SMOVL C00364 BC00364 V=166.7  +MOVJ EC00364
SREFP 3 C00365 BC00365  +REFP EC00365
CALL JOB:SEARCH-R1-S13D
SET P028 P006
SFTON3D P028
SMOVL C00366 BC00366 V=166.7  +MOVJ EC00366
SREFP 3 C00367 BC00367  +REFP EC00367
CALL JOB:SEARCH-R1-S13D
SET P028 P006
SFTON3D P028
SMOVL C00368 BC00368 V=250.0  +MOVJ EC00368
MOVL C00369 BC00369 V=1000.0  +MOVJ EC00369 VJ=100.00
'EndPath S4609
MOVJ C00370 BC00370 VJ=100.00  +MOVJ EC00370 VJ=100.00
'Path S4882
SFTOF3D
MOVJ C00371 BC00371 VJ=100.00  +MOVJ EC00371 VJ=100.00
MOVL C00372 BC00372 V=800.0  +MOVJ EC00372 VJ=100.00
SMOVL C00373 BC00373 V=166.7  +MOVJ EC00373
SREFP 3 C00374 BC00374  +REFP EC00374
CALL JOB:SEARCH-R1-S13D
SET P060 P006
SFTON3D P060
SMOVL C00375 BC00375 V=166.7  +MOVJ EC00375
SMOVL C00376 BC00376 V=166.7  +MOVJ EC00376
SREFP 3 C00377 BC00377  +REFP EC00377
CALL JOB:SEARCH-R1-S13D
SET P060 P006
SFTON3D P060
SMOVL C00378 BC00378 V=166.7  +MOVJ EC00378
SMOVL C00379 BC00379 V=333.3  +MOVJ EC00379
SMOVL C00380 BC00380 V=166.7  +MOVJ EC00380
SREFP 3 C00381 BC00381  +REFP EC00381
CALL JOB:SEARCH-R1-S13D
SET P060 P006
SFTON3D P060
SMOVL C00382 BC00382 V=166.7  +MOVJ EC00382
MOVL C00383 BC00383 V=1000.0  +MOVJ EC00383 VJ=100.00
'EndPath S4882
MOVJ C00384 BC00384 VJ=100.00  +MOVJ EC00384 VJ=100.00
COMM 'Path S4610
COMM PAUSE
COMM SFTOF3D
COMM MOVJ C00385 BC00385 VJ=100.00  +MOVJ EC00385 VJ=100.00
COMM MOVL C00386 BC00386 V=800.0  +MOVJ EC00386 VJ=100.00
COMM SMOVL C00387 BC00387 V=166.7  +MOVJ EC00387
COMM SREFP 3 C00388 BC00388  +REFP EC00388
COMM CALL JOB:SEARCH-R1-S13D
COMM SET P029 P006
COMM SFTON3D P029
COMM SMOVL C00389 BC00389 V=166.7  +MOVJ EC00389
COMM SREFP 3 C00390 BC00390  +REFP EC00390
COMM CALL JOB:SEARCH-R1-S13D
COMM SET P029 P006
COMM SFTON3D P029
COMM SMOVL C00391 BC00391 V=166.7  +MOVJ EC00391
COMM MOVL C00392 BC00392 V=1000.0  +MOVJ EC00392 VJ=100.00
COMM 'EndPath S4610
COMM 'Path S4611
COMM SFTOF3D
COMM MOVJ C00393 BC00393 VJ=100.00  +MOVJ EC00393 VJ=100.00
COMM MOVL C00394 BC00394 V=800.0  +MOVJ EC00394 VJ=100.00
COMM SMOVL C00395 BC00395 V=166.7  +MOVJ EC00395
COMM SREFP 3 C00396 BC00396  +REFP EC00396
COMM CALL JOB:SEARCH-R1-S13D
COMM SET P030 P006
COMM SFTON3D P030
COMM SMOVL C00397 BC00397 V=166.7  +MOVJ EC00397
COMM SREFP 3 C00398 BC00398  +REFP EC00398
COMM CALL JOB:SEARCH-R1-S13D
COMM SET P030 P006
COMM SFTON3D P030
COMM SMOVL C00399 BC00399 V=166.7  +MOVJ EC00399
COMM MOVL C00400 BC00400 V=800.0  +MOVJ EC00400 VJ=100.00
COMM MOVL C00401 BC00401 V=1000.0  +MOVJ EC00401 VJ=100.00
COMM 'EndPath S4611
MOVJ C00402 BC00402 VJ=100.00  +MOVJ EC00402 VJ=100.00
'Path S4612
SFTOF3D
MOVJ C00403 BC00403 VJ=100.00  +MOVJ EC00403 VJ=100.00
MOVL C00404 BC00404 V=800.0  +MOVJ EC00404 VJ=100.00
SMOVL C00405 BC00405 V=166.7  +MOVJ EC00405
SREFP 3 C00406 BC00406  +REFP EC00406
CALL JOB:SEARCH-R1-S13D
SET P031 P006
SFTON3D P031
SMOVL C00407 BC00407 V=166.7  +MOVJ EC00407
SMOVL C00408 BC00408 V=166.7  +MOVJ EC00408
SREFP 3 C00409 BC00409  +REFP EC00409
CALL JOB:SEARCH-R1-S13D
SET P031 P006
SFTON3D P031
SMOVL C00410 BC00410 V=166.7  +MOVJ EC00410
SMOVL C00411 BC00411 V=166.7  +MOVJ EC00411
SREFP 3 C00412 BC00412  +REFP EC00412
CALL JOB:SEARCH-R1-S13D
SET P031 P006
SFTON3D P031
SMOVL C00413 BC00413 V=166.7  +MOVJ EC00413
MOVL C00414 BC00414 V=1000.0  +MOVJ EC00414 VJ=100.00
'EndPath S4612
MOVJ C00415 BC00415 VJ=100.00  +MOVJ EC00415 VJ=100.00
'Path S4613
SFTOF3D
MOVJ C00416 BC00416 VJ=100.00  +MOVJ EC00416 VJ=100.00
MOVL C00417 BC00417 V=800.0  +MOVJ EC00417 VJ=100.00
SMOVL C00418 BC00418 V=166.7  +MOVJ EC00418
SREFP 3 C00419 BC00419  +REFP EC00419
CALL JOB:SEARCH-R1-S13D
SET P032 P006
SFTON3D P032
SMOVL C00420 BC00420 V=166.7  +MOVJ EC00420
SREFP 3 C00421 BC00421  +REFP EC00421
CALL JOB:SEARCH-R1-S13D
SET P032 P006
SFTON3D P032
SMOVL C00422 BC00422 V=166.7  +MOVJ EC00422
SMOVL C00423 BC00423 V=166.7  +MOVJ EC00423
SREFP 3 C00424 BC00424  +REFP EC00424
CALL JOB:SEARCH-R1-S13D
SET P032 P006
SFTON3D P032
SMOVL C00425 BC00425 V=166.7  +MOVJ EC00425
MOVL C00426 BC00426 V=1000.0  +MOVJ EC00426 VJ=100.00
'EndPath S4613
MOVJ C00427 BC00427 VJ=100.00  +MOVJ EC00427 VJ=100.00
'Path S4614
SFTOF3D
MOVJ C00428 BC00428 VJ=100.00  +MOVJ EC00428 VJ=100.00
MOVL C00429 BC00429 V=800.0  +MOVJ EC00429 VJ=100.00
SMOVL C00430 BC00430 V=166.7  +MOVJ EC00430
SREFP 3 C00431 BC00431  +REFP EC00431
CALL JOB:SEARCH-R1-S13D
SET P033 P006
SFTON3D P033
SMOVL C00432 BC00432 V=166.7  +MOVJ EC00432
SREFP 3 C00433 BC00433  +REFP EC00433
CALL JOB:SEARCH-R1-S13D
SET P033 P006
SFTON3D P033
SMOVL C00434 BC00434 V=166.7  +MOVJ EC00434
MOVL C00435 BC00435 V=1000.0  +MOVJ EC00435 VJ=100.00
'EndPath S4614
'Path S4615
SFTOF3D
MOVJ C00436 BC00436 VJ=100.00  +MOVJ EC00436 VJ=100.00
MOVL C00437 BC00437 V=800.0  +MOVJ EC00437 VJ=100.00
SMOVL C00438 BC00438 V=166.7  +MOVJ EC00438
SREFP 3 C00439 BC00439  +REFP EC00439
CALL JOB:SEARCH-R1-S13D
SET P034 P006
SFTON3D P034
SMOVL C00440 BC00440 V=166.7  +MOVJ EC00440
SREFP 3 C00441 BC00441  +REFP EC00441
CALL JOB:SEARCH-R1-S13D
SET P034 P006
SFTON3D P034
SMOVL C00442 BC00442 V=166.7  +MOVJ EC00442
SMOVL C00443 BC00443 V=166.7  +MOVJ EC00443
SREFP 3 C00444 BC00444  +REFP EC00444
CALL JOB:SEARCH-R1-S13D
SET P034 P006
SFTON3D P034
SMOVL C00445 BC00445 V=166.7  +MOVJ EC00445
MOVL C00446 BC00446 V=1000.0  +MOVJ EC00446 VJ=100.00
'EndPath S4615
MOVJ C00447 BC00447 VJ=100.00  +MOVJ EC00447 VJ=100.00
MOVJ C00448 BC00448 VJ=100.00  +MOVJ EC00448 VJ=100.00
'Path W4616
SFTOF3D
SFTON3D P026
MOVJ C00449 BC00449 VJ=100.00  +MOVJ EC00449 VJ=100.00
SMOVL C00450 BC00450 V=800.0  +MOVJ EC00450
'POPRAWIC!!!!
SMOVL C00451 BC00451 V=166.7 PL=0  +MOVJ EC00451
MACRO1 MJ#(0) ARGF21
ARCON
SWVON WEV#(100)
SMOVL C00452 BC00452 V=9.2  +MOVJ EC00452
SFTON3D P091
SMOVL C00453 BC00453 V=9.2  +MOVJ EC00453
SMOVL C00454 BC00454 V=9.2  +MOVJ EC00454
SWVOF
ARCOF
SMOVL C00455 BC00455 V=800.0  +MOVJ EC00455
SMOVL C00456 BC00456 V=1000.0  +MOVJ EC00456
SFTOF3D
'EndPath W4616
MOVJ C00457 BC00457 VJ=100.00  +MOVJ EC00457 VJ=100.00
'Path W4617
SFTOF3D
SFTON3D P028
MOVJ C00458 BC00458 VJ=100.00  +MOVJ EC00458 VJ=100.00
MOVJ C00459 BC00459 VJ=100.00  +MOVJ EC00459 VJ=100.00
SMOVL C00460 BC00460 V=800.0  +MOVJ EC00460
SMOVL C00461 BC00461 V=150.0 PL=0  +MOVJ EC00461
ARCON
SWVON WEV#(100)
MOVL C00462 BC00462 V=9.2  +MOVJ EC00462 VJ=100.00
SFTON3D P027
SMOVL C00463 BC00463 V=9.2  +MOVJ EC00463
SMOVL C00464 BC00464 V=9.2  +MOVJ EC00464
ARCOF
SWVOF
SMOVL C00465 BC00465 V=800.0  +MOVJ EC00465
SMOVL C00466 BC00466 V=1000.0  +MOVJ EC00466
SFTOF3D
'EndPath W4617
MOVJ C00467 BC00467 VJ=100.00  +MOVJ EC00467 VJ=100.00
'Path W4618
COMM PAUSE
COMM SFTOF3D
COMM SFTON3D P022
COMM MOVJ C00468 BC00468 VJ=100.00  +MOVJ EC00468 VJ=100.00
COMM SMOVL C00469 BC00469 V=800.0  +MOVJ EC00469
COMM SMOVL C00470 BC00470 V=150.0 PL=0  +MOVJ EC00470
COMM MACRO1 MJ#(0) ARGF9
COMM ARCON
COMM SWVON WEV#(60)
COMM SFTON3D P021
COMM SMOVL C00471 BC00471 V=10.0  +MOVJ EC00471
COMM ARCOF
COMM SWVOF
COMM SMOVL C00472 BC00472 V=800.0  +MOVJ EC00472
COMM SMOVL C00473 BC00473 V=1000.0  +MOVJ EC00473
COMM SFTOF3D
COMM 'EndPath W4618
COMM 'Path W4883
SFTOF3D
SFTON3D P060
MOVJ C00474 BC00474 VJ=100.00  +MOVJ EC00474 VJ=100.00
MACRO1 MJ#(0) ARGF9
SMOVL C00475 BC00475 V=800.0  +MOVJ EC00475
SMOVL C00476 BC00476 V=150.0 PL=0  +MOVJ EC00476
ARCON
SMOVL C00477 BC00477 V=10.0  +MOVJ EC00477
SMOVL C00478 BC00478 V=10.0  +MOVJ EC00478
SMOVL C00479 BC00479 V=10.0  +MOVJ EC00479
ARCOF
SMOVL C00480 BC00480 V=800.0  +MOVJ EC00480
SFTOF3D
'EndPath W4883
'Path W4884
SFTOF3D
SFTON3D P060
SMOVL C00481 BC00481 V=800.0  +MOVJ EC00481
SMOVL C00482 BC00482 V=150.0 PL=0  +MOVJ EC00482
ARCON
SMOVL C00483 BC00483 V=10.0  +MOVJ EC00483
SMOVL C00484 BC00484 V=10.0  +MOVJ EC00484
SMOVL C00485 BC00485 V=10.0  +MOVJ EC00485
ARCOF
SMOVL C00486 BC00486 V=800.0  +MOVJ EC00486
SMOVL C00487 BC00487 V=1000.0  +MOVJ EC00487
SFTOF3D
'EndPath W4884
MOVJ C00488 BC00488 VJ=100.00  +MOVJ EC00488 VJ=100.00
COMM 'Path W4619
COMM PAUSE
COMM SFTOF3D
COMM SFTON3D P030
COMM MOVJ C00489 BC00489 VJ=100.00  +MOVJ EC00489 VJ=100.00
COMM MOVJ C00490 BC00490 VJ=100.00  +MOVJ EC00490 VJ=100.00
COMM SMOVL C00491 BC00491 V=800.0  +MOVJ EC00491
COMM SMOVL C00492 BC00492 V=150.0 PL=0  +MOVJ EC00492
COMM ARCON
COMM MOVL C00493 BC00493 V=10.0  +MOVJ EC00493 VJ=100.00
COMM SFTON3D P029
COMM SMOVL C00494 BC00494 V=10.0  +MOVJ EC00494
COMM SMOVL C00495 BC00495 V=10.0  +MOVJ EC00495
COMM ARCOF
COMM SMOVL C00496 BC00496 V=800.0  +MOVJ EC00496
COMM SMOVL C00497 BC00497 V=1000.0  +MOVJ EC00497
COMM SFTOF3D
COMM 'EndPath W4619
MOVJ C00498 BC00498 VJ=100.00  +MOVJ EC00498 VJ=100.00
MOVJ C00499 BC00499 VJ=100.00  +MOVJ EC00499 VJ=100.00
'Path W4620
SFTOF3D
SFTON3D P033
MOVJ C00500 BC00500 VJ=100.00  +MOVJ EC00500 VJ=100.00
SMOVL C00501 BC00501 V=800.0  +MOVJ EC00501
SMOVL C00502 BC00502 V=166.7 PL=0  +MOVJ EC00502
ARCON
SMOVL C00503 BC00503 V=9.2  +MOVJ EC00503
SFTON3D P034
SMOVL C00504 BC00504 V=9.2  +MOVJ EC00504
SMOVL C00505 BC00505 V=9.2  +MOVJ EC00505
ARCOF
SMOVL C00506 BC00506 V=800.0  +MOVJ EC00506
SMOVL C00507 BC00507 V=1000.0  +MOVJ EC00507
SFTOF3D
'EndPath W4620
MOVJ C00508 BC00508 VJ=100.00  +MOVJ EC00508 VJ=100.00
'Path W4621
SFTOF3D
SFTON3D P024
MOVJ C00509 BC00509 VJ=100.00  +MOVJ EC00509 VJ=100.00
SMOVL C00510 BC00510 V=800.0  +MOVJ EC00510
SMOVL C00511 BC00511 V=166.7 PL=0  +MOVJ EC00511
ARCON
SMOVL C00512 BC00512 V=10.0  +MOVJ EC00512
SFTON3D P025
SMOVL C00513 BC00513 V=10.0  +MOVJ EC00513
SMOVL C00514 BC00514 V=10.0  +MOVJ EC00514
ARCOF
SMOVL C00515 BC00515 V=800.0  +MOVJ EC00515
SMOVL C00516 BC00516 V=1000.0  +MOVJ EC00516
SFTOF3D
'EndPath W4621
MOVJ C00517 BC00517 VJ=100.00  +MOVJ EC00517 VJ=100.00
MOVJ C00518 BC00518 VJ=100.00  +MOVJ EC00518 VJ=100.00
'Path W4622
SFTOF3D
SFTON3D P032
MOVJ C00519 BC00519 VJ=100.00  +MOVJ EC00519 VJ=100.00
SMOVL C00520 BC00520 V=800.0  +MOVJ EC00520
SMOVL C00521 BC00521 V=166.7 PL=0  +MOVJ EC00521
ARCON
SMOVL C00522 BC00522 V=9.2  +MOVJ EC00522
SFTON3D P031
SMOVL C00523 BC00523 V=9.2  +MOVJ EC00523
SMOVL C00524 BC00524 V=9.2  +MOVJ EC00524
ARCOF
SMOVL C00525 BC00525 V=800.0  +MOVJ EC00525
SMOVL C00526 BC00526 V=1000.0  +MOVJ EC00526
SFTOF3D
'EndPath W4622
'Path W4623
SFTOF3D
SFTON3D P023
MOVJ C00527 BC00527 VJ=100.00  +MOVJ EC00527 VJ=100.00
JUMP *VVP
MOVJ C00528 BC00528 VJ=100.00  +MOVJ EC00528 VJ=100.00
SMOVL C00529 BC00529 V=800.0  +MOVJ EC00529
SMOVL C00530 BC00530 V=166.7 PL=0  +MOVJ EC00530
'ARCON DO SPRAWDZENIA
PAUSE
SMOVL C00531 BC00531 V=10.0  +MOVJ EC00531
SMOVL C00532 BC00532 V=10.0  +MOVJ EC00532
SMOVL C00533 BC00533 V=10.0  +MOVJ EC00533
SMOVL C00534 BC00534 V=10.0  +MOVJ EC00534
SMOVL C00535 BC00535 V=10.0  +MOVJ EC00535
SMOVL C00536 BC00536 V=10.0  +MOVJ EC00536
SMOVL C00537 BC00537 V=10.0  +MOVJ EC00537
SMOVL C00538 BC00538 V=10.0  +MOVJ EC00538
SMOVL C00539 BC00539 V=10.0  +MOVJ EC00539
ARCOF
SMOVL C00540 BC00540 V=800.0  +MOVJ EC00540
SMOVL C00541 BC00541 V=1000.0  +MOVJ EC00541
SFTOF3D
'EndPath W4623
'Path W4624
*VVP
MOVJ C00542 BC00542 VJ=100.00  +MOVJ EC00542 VJ=100.00
SFTOF3D
SFTON3D P023
MOVJ C00543 BC00543 VJ=100.00  +MOVJ EC00543 VJ=100.00
SMOVL C00544 BC00544 V=800.0  +MOVJ EC00544
COMM SMOVL C00545 BC00545 V=150.0 PL=0  +MOVJ EC00545
COMM ARCON
COMM SMOVL C00546 BC00546 V=8.3  +MOVJ EC00546
SMOVL C00547 BC00547 V=166.7 PL=0  +MOVJ EC00547
ARCON
SMOVL C00548 BC00548 V=8.3  +MOVJ EC00548
SMOVL C00549 BC00549 V=8.3  +MOVJ EC00549
SMOVL C00550 BC00550 V=8.3  +MOVJ EC00550
SMOVL C00551 BC00551 V=8.3  +MOVJ EC00551
MOVL C00552 BC00552 V=8.3  +MOVJ EC00552 VJ=100.00
ARCOF
SMOVL C00553 BC00553 V=800.0  +MOVJ EC00553
SMOVL C00554 BC00554 V=1000.0  +MOVJ EC00554
SFTOF3D
'EndPath W4624
MOVJ C00555 BC00555 VJ=100.00  +MOVJ EC00555 VJ=100.00
'Path S4625
SFTOF3D
CALL JOB:CLEAN-R1_KM_3P
MOVJ C00556 BC00556 VJ=100.00  +MOVJ EC00556 VJ=100.00
MOVJ C00557 BC00557 VJ=100.00  +MOVJ EC00557 VJ=100.00
MOVL C00558 BC00558 V=800.0  +MOVJ EC00558 VJ=100.00
SMOVL C00559 BC00559 V=166.7  +MOVJ EC00559
SREFP 3 C00560 BC00560  +REFP EC00560
CALL JOB:SEARCH-R1-S13D
SET P048 P006
SFTON3D P048
SMOVL C00561 BC00561 V=166.7  +MOVJ EC00561
SMOVL C00562 BC00562 V=166.7  +MOVJ EC00562
SREFP 3 C00563 BC00563  +REFP EC00563
CALL JOB:SEARCH-R1-S13D
SET P048 P006
SFTON3D P048
SMOVL C00564 BC00564 V=16.7  +MOVJ EC00564
MOVL C00565 BC00565 V=800.0  +MOVJ EC00565 VJ=100.00
MOVL C00566 BC00566 V=1000.0  +MOVJ EC00566 VJ=100.00
'EndPath S4625
'Path S4626
SFTOF3D
MOVJ C00567 BC00567 VJ=100.00  +MOVJ EC00567 VJ=100.00
MOVL C00568 BC00568 V=800.0  +MOVJ EC00568 VJ=100.00
SMOVL C00569 BC00569 V=166.7  +MOVJ EC00569
SREFP 3 C00570 BC00570  +REFP EC00570
CALL JOB:SEARCH-R1-S13D
SET P047 P006
SFTON3D P047
SMOVL C00571 BC00571 V=166.7  +MOVJ EC00571
SMOVL C00572 BC00572 V=166.7  +MOVJ EC00572
SREFP 3 C00573 BC00573  +REFP EC00573
CALL JOB:SEARCH-R1-S13D
SET P047 P006
SFTON3D P047
SMOVL C00574 BC00574 V=166.7  +MOVJ EC00574
MOVL C00575 BC00575 V=800.0  +MOVJ EC00575 VJ=100.00
MOVL C00576 BC00576 V=1000.0  +MOVJ EC00576 VJ=100.00
'EndPath S4626
MOVJ C00577 BC00577 VJ=100.00  +MOVJ EC00577 VJ=100.00
'Path S4627
SFTOF3D
MOVJ C00578 BC00578 VJ=100.00  +MOVJ EC00578 VJ=100.00
MOVL C00579 BC00579 V=800.0  +MOVJ EC00579 VJ=100.00
SMOVL C00580 BC00580 V=166.7  +MOVJ EC00580
SREFP 3 C00581 BC00581  +REFP EC00581
CALL JOB:SEARCH-R1-S13D
SET P046 P006
SFTON3D P046
SMOVL C00582 BC00582 V=166.7  +MOVJ EC00582
MOVL C00583 BC00583 V=800.0  +MOVJ EC00583 VJ=100.00
SMOVL C00584 BC00584 V=166.7  +MOVJ EC00584
SREFP 3 C00585 BC00585  +REFP EC00585
CALL JOB:SEARCH-R1-S13D
SET P046 P006
SFTON3D P046
SMOVL C00586 BC00586 V=166.7  +MOVJ EC00586
MOVL C00587 BC00587 V=800.0  +MOVJ EC00587 VJ=100.00
MOVL C00588 BC00588 V=1000.0  +MOVJ EC00588 VJ=100.00
'EndPath S4627
'Path S4628
SFTOF3D
MOVJ C00589 BC00589 VJ=100.00  +MOVJ EC00589 VJ=100.00
MOVL C00590 BC00590 V=800.0  +MOVJ EC00590 VJ=100.00
SMOVL C00591 BC00591 V=166.7  +MOVJ EC00591
SREFP 3 C00592 BC00592  +REFP EC00592
CALL JOB:SEARCH-R1-S13D
SET P050 P006
SFTON3D P050
SMOVL C00593 BC00593 V=166.7  +MOVJ EC00593
SMOVL C00594 BC00594 V=800.0  +MOVJ EC00594
SMOVL C00595 BC00595 V=166.7  +MOVJ EC00595
SREFP 3 C00596 BC00596  +REFP EC00596
CALL JOB:SEARCH-R1-S13D
SET P050 P006
SFTON3D P050
SMOVL C00597 BC00597 V=166.7  +MOVJ EC00597
MOVL C00598 BC00598 V=800.0  +MOVJ EC00598 VJ=100.00
MOVL C00599 BC00599 V=1000.0  +MOVJ EC00599 VJ=100.00
'EndPath S4628
'Path S4629
SFTOF3D
MOVJ C00600 BC00600 VJ=100.00  +MOVJ EC00600 VJ=100.00
MOVJ C00601 BC00601 VJ=100.00  +MOVJ EC00601 VJ=100.00
MOVL C00602 BC00602 V=800.0  +MOVJ EC00602 VJ=100.00
SMOVL C00603 BC00603 V=166.7  +MOVJ EC00603
SREFP 3 C00604 BC00604  +REFP EC00604
CALL JOB:SEARCH-R1-S13D
SET P051 P006
SFTON3D P051
SMOVL C00605 BC00605 V=166.7  +MOVJ EC00605
SREFP 3 C00606 BC00606  +REFP EC00606
CALL JOB:SEARCH-R1-S13D
SET P051 P006
SFTON3D P051
SMOVL C00607 BC00607 V=166.7  +MOVJ EC00607
SMOVL C00608 BC00608 V=250.0  +MOVJ EC00608
SMOVL C00609 BC00609 V=166.7  +MOVJ EC00609
SREFP 3 C00610 BC00610  +REFP EC00610
CALL JOB:SEARCH-R1-S13D
SET P051 P006
SFTON3D P051
SMOVL C00611 BC00611 V=166.7  +MOVJ EC00611
MOVL C00612 BC00612 V=1000.0  +MOVJ EC00612 VJ=100.00
'EndPath S4629
'Path S4630
SFTOF3D
MOVJ C00613 BC00613 VJ=100.00  +MOVJ EC00613 VJ=100.00
MOVL C00614 BC00614 V=800.0  +MOVJ EC00614 VJ=100.00
SMOVL C00615 BC00615 V=166.7  +MOVJ EC00615
SREFP 3 C00616 BC00616  +REFP EC00616
CALL JOB:SEARCH-R1-S13D
SET P045 P006
SFTON3D P045
SMOVL C00617 BC00617 V=166.7  +MOVJ EC00617
SMOVL C00618 BC00618 V=166.7  +MOVJ EC00618
SREFP 3 C00619 BC00619  +REFP EC00619
CALL JOB:SEARCH-R1-S13D
SET P045 P006
SFTON3D P045
SMOVL C00620 BC00620 V=166.7  +MOVJ EC00620
MOVL C00621 BC00621 V=1000.0  +MOVJ EC00621 VJ=100.00
'EndPath S4630
'Path S4631
SFTOF3D
MOVJ C00622 BC00622 VJ=100.00  +MOVJ EC00622 VJ=100.00
MOVL C00623 BC00623 V=800.0  +MOVJ EC00623 VJ=100.00
SMOVL C00624 BC00624 V=166.7  +MOVJ EC00624
SREFP 3 C00625 BC00625  +REFP EC00625
CALL JOB:SEARCH-R1-S13D
SET P044 P006
SFTON3D P044
SMOVL C00626 BC00626 V=166.7  +MOVJ EC00626
SMOVL C00627 BC00627 V=166.7  +MOVJ EC00627
SREFP 3 C00628 BC00628  +REFP EC00628
CALL JOB:SEARCH-R1-S13D
SET P044 P006
SFTON3D P044
SMOVL C00629 BC00629 V=166.7  +MOVJ EC00629
MOVL C00630 BC00630 V=800.0  +MOVJ EC00630 VJ=100.00
MOVL C00631 BC00631 V=1000.0  +MOVJ EC00631 VJ=100.00
'EndPath S4631
'Path S4632
SFTOF3D
MOVJ C00632 BC00632 VJ=100.00  +MOVJ EC00632 VJ=100.00
MOVL C00633 BC00633 V=800.0  +MOVJ EC00633 VJ=100.00
SMOVL C00634 BC00634 V=166.7  +MOVJ EC00634
SREFP 3 C00635 BC00635  +REFP EC00635
CALL JOB:SEARCH-R1-S13D
SET P049 P006
SFTON3D P049
SMOVL C00636 BC00636 V=166.7  +MOVJ EC00636
SMOVL C00637 BC00637 V=800.0  +MOVJ EC00637
SMOVL C00638 BC00638 V=166.7  +MOVJ EC00638
SREFP 3 C00639 BC00639  +REFP EC00639
CALL JOB:SEARCH-R1-S13D
SET P049 P006
SFTON3D P049
SMOVL C00640 BC00640 V=166.7  +MOVJ EC00640
MOVL C00641 BC00641 V=1000.0  +MOVJ EC00641 VJ=100.00
'EndPath S4632
MOVJ C00642 BC00642 VJ=100.00  +MOVJ EC00642 VJ=100.00
MOVJ C00643 BC00643 VJ=100.00  +MOVJ EC00643 VJ=100.00
MOVJ C00644 BC00644 VJ=100.00  +MOVJ EC00644 VJ=100.00
MOVJ C00645 BC00645 VJ=100.00  +MOVJ EC00645 VJ=100.00
'Path S4633
SFTOF3D
MOVJ C00646 BC00646 VJ=100.00  +MOVJ EC00646 VJ=100.00
MOVL C00647 BC00647 V=800.0  +MOVJ EC00647 VJ=100.00
SMOVL C00648 BC00648 V=166.7  +MOVJ EC00648
SREFP 3 C00649 BC00649  +REFP EC00649
CALL JOB:SEARCH-R1-S13D
SET P043 P006
SFTON3D P043
SMOVL C00650 BC00650 V=166.7  +MOVJ EC00650
MOVL C00651 BC00651 V=800.0  +MOVJ EC00651 VJ=100.00
SMOVL C00652 BC00652 V=166.7  +MOVJ EC00652
SREFP 3 C00653 BC00653  +REFP EC00653
CALL JOB:SEARCH-R1-S13D
SET P043 P006
SFTON3D P043
SMOVL C00654 BC00654 V=166.7  +MOVJ EC00654
MOVL C00655 BC00655 V=1000.0  +MOVJ EC00655 VJ=100.00
'EndPath S4633
'Path S4634
SFTOF3D
MOVJ C00656 BC00656 VJ=100.00  +MOVJ EC00656 VJ=100.00
MOVL C00657 BC00657 V=800.0  +MOVJ EC00657 VJ=100.00
SMOVL C00658 BC00658 V=166.7  +MOVJ EC00658
SREFP 3 C00659 BC00659  +REFP EC00659
CALL JOB:SEARCH-R1-S13D
SET P042 P006
SFTON3D P042
SMOVL C00660 BC00660 V=166.7  +MOVJ EC00660
MOVL C00661 BC00661 V=800.0  +MOVJ EC00661 VJ=100.00
SMOVL C00662 BC00662 V=166.7  +MOVJ EC00662
SREFP 3 C00663 BC00663  +REFP EC00663
CALL JOB:SEARCH-R1-S13D
SET P042 P006
SFTON3D P042
SMOVL C00664 BC00664 V=166.7  +MOVJ EC00664
MOVL C00665 BC00665 V=1000.0  +MOVJ EC00665 VJ=100.00
'EndPath S4634
MOVJ C00666 BC00666 VJ=100.00  +MOVJ EC00666 VJ=100.00
MOVJ C00667 BC00667 VJ=100.00  +MOVJ EC00667 VJ=100.00
MOVJ C00668 BC00668 VJ=100.00  +MOVJ EC00668 VJ=100.00
MOVJ C00669 BC00669 VJ=100.00  +MOVJ EC00669 VJ=100.00
'Path W4635
SFTOF3D
SFTON3D P051
MOVJ C00670 BC00670 VJ=100.00  +MOVJ EC00670 VJ=100.00
SMOVL C00671 BC00671 V=800.0  +MOVJ EC00671
SMOVL C00672 BC00672 V=150.0 PL=0  +MOVJ EC00672
MACRO1 MJ#(0) ARGF14
ARCON
SMOVL C00673 BC00673 V=11.7  +MOVJ EC00673
ARCOF
SMOVL C00674 BC00674 V=800.0  +MOVJ EC00674
SMOVL C00675 BC00675 V=1000.0  +MOVJ EC00675
MOVJ C00676 BC00676 VJ=100.00  +MOVJ EC00676 VJ=100.00
MOVJ C00677 BC00677 VJ=100.00  +MOVJ EC00677 VJ=100.00
SMOVL C00678 BC00678 V=250.0  +MOVJ EC00678
ARCON
SMOVL C00679 BC00679 V=11.7  +MOVJ EC00679
SMOVL C00680 BC00680 V=11.7  +MOVJ EC00680
ARCOF
SMOVL C00681 BC00681 V=166.7  +MOVJ EC00681
SMOVL C00682 BC00682 V=166.7  +MOVJ EC00682
SMOVL C00683 BC00683 V=166.7  +MOVJ EC00683
ARCON
SMOVL C00684 BC00684 V=9.2  +MOVJ EC00684
ARCOF
SMOVL C00685 BC00685 V=133.3  +MOVJ EC00685
SMOVL C00686 BC00686 V=666.7  +MOVJ EC00686
SFTOF3D
'EndPath W4635
'Path W4636
SFTOF3D
SFTON3D P045
MOVJ C00687 BC00687 VJ=100.00  +MOVJ EC00687 VJ=100.00
SMOVL C00688 BC00688 V=800.0  +MOVJ EC00688
SMOVL C00689 BC00689 V=150.0 PL=0  +MOVJ EC00689
MACRO1 MJ#(0) ARGF21
ARCON
SMOVL C00690 BC00690 V=11.7  +MOVJ EC00690
SMOVL C00691 BC00691 V=11.7  +MOVJ EC00691
ARCOF
SMOVL C00692 BC00692 V=800.0  +MOVJ EC00692
SMOVL C00693 BC00693 V=1000.0  +MOVJ EC00693
SFTOF3D
'EndPath W4636
'Path W4637
SFTOF3D
SFTON3D P045
MOVJ C00694 BC00694 VJ=100.00  +MOVJ EC00694 VJ=100.00
SMOVL C00695 BC00695 V=800.0  +MOVJ EC00695
SMOVL C00696 BC00696 V=150.0 PL=0  +MOVJ EC00696
ARCON
SMOVL C00697 BC00697 V=11.7  +MOVJ EC00697
SMOVL C00698 BC00698 V=11.7  +MOVJ EC00698
ARCOF
SMOVL C00699 BC00699 V=800.0  +MOVJ EC00699
SMOVL C00700 BC00700 V=1000.0  +MOVJ EC00700
SFTOF3D
'EndPath W4637
'Path W4638
SFTOF3D
SFTON3D P049
MOVJ C00701 BC00701 VJ=100.00  +MOVJ EC00701 VJ=100.00
SMOVL C00702 BC00702 V=800.0  +MOVJ EC00702
SMOVL C00703 BC00703 V=150.0 PL=0  +MOVJ EC00703
ARCON
SMOVL C00704 BC00704 V=10.0  +MOVJ EC00704
ARCOF
SMOVL C00705 BC00705 V=800.0  +MOVJ EC00705
SMOVL C00706 BC00706 V=1000.0  +MOVJ EC00706
SFTOF3D
'EndPath W4638
'Path W4639
SFTOF3D
SFTON3D P050
MOVJ C00707 BC00707 VJ=100.00  +MOVJ EC00707 VJ=100.00
SMOVL C00708 BC00708 V=800.0  +MOVJ EC00708
SMOVL C00709 BC00709 V=150.0 PL=0  +MOVJ EC00709
ARCON
SMOVL C00710 BC00710 V=11.7  +MOVJ EC00710
ARCOF
SMOVL C00711 BC00711 V=800.0  +MOVJ EC00711
SMOVL C00712 BC00712 V=1000.0  +MOVJ EC00712
SFTOF3D
'EndPath W4639
MOVJ C00713 BC00713 VJ=100.00  +MOVJ EC00713 VJ=100.00
'Path W4640
SFTOF3D
SFTON3D P048
MOVJ C00714 BC00714 VJ=100.00  +MOVJ EC00714 VJ=100.00
SMOVL C00715 BC00715 V=800.0  +MOVJ EC00715
SMOVL C00716 BC00716 V=150.0 PL=0  +MOVJ EC00716
ARCON
SMOVL C00717 BC00717 V=11.7  +MOVJ EC00717
ARCOF
SMOVL C00718 BC00718 V=800.0  +MOVJ EC00718
SMOVL C00719 BC00719 V=1000.0  +MOVJ EC00719
SFTOF3D
'EndPath W4640
'Path W4641
SFTOF3D
SFTON3D P048
MOVJ C00720 BC00720 VJ=100.00  +MOVJ EC00720 VJ=100.00
SMOVL C00721 BC00721 V=800.0  +MOVJ EC00721
SMOVL C00722 BC00722 V=150.0 PL=0  +MOVJ EC00722
ARCON
SMOVL C00723 BC00723 V=11.7  +MOVJ EC00723
ARCOF
SMOVL C00724 BC00724 V=800.0  +MOVJ EC00724
SMOVL C00725 BC00725 V=1000.0  +MOVJ EC00725
SFTOF3D
'EndPath W4641
'Path W4642
SFTOF3D
SFTON3D P047
MOVJ C00726 BC00726 VJ=100.00  +MOVJ EC00726 VJ=100.00
SMOVL C00727 BC00727 V=800.0  +MOVJ EC00727
SMOVL C00728 BC00728 V=150.0 PL=0  +MOVJ EC00728
ARCON
SMOVL C00729 BC00729 V=11.7  +MOVJ EC00729
ARCOF
SMOVL C00730 BC00730 V=800.0  +MOVJ EC00730
SMOVL C00731 BC00731 V=1000.0  +MOVJ EC00731
SFTOF3D
'EndPath W4642
MOVJ C00732 BC00732 VJ=100.00  +MOVJ EC00732 VJ=100.00
MOVJ C00733 BC00733 VJ=100.00  +MOVJ EC00733 VJ=100.00
'Path W4643
SFTOF3D
SFTON3D P043
MOVJ C00734 BC00734 VJ=100.00  +MOVJ EC00734 VJ=100.00
SMOVL C00735 BC00735 V=800.0  +MOVJ EC00735
SMOVL C00736 BC00736 V=150.0 PL=0  +MOVJ EC00736
ARCON
SMOVL C00737 BC00737 V=11.7  +MOVJ EC00737
ARCOF
SMOVL C00738 BC00738 V=800.0  +MOVJ EC00738
SMOVL C00739 BC00739 V=1000.0  +MOVJ EC00739
SFTOF3D
'EndPath W4643
'Path W4644
SFTOF3D
SFTON3D P043
MOVJ C00740 BC00740 VJ=100.00  +MOVJ EC00740 VJ=100.00
SMOVL C00741 BC00741 V=800.0  +MOVJ EC00741
SMOVL C00742 BC00742 V=150.0 PL=0  +MOVJ EC00742
ARCON
SMOVL C00743 BC00743 V=11.7  +MOVJ EC00743
ARCOF
SMOVL C00744 BC00744 V=800.0  +MOVJ EC00744
SMOVL C00745 BC00745 V=1000.0  +MOVJ EC00745
SFTOF3D
'EndPath W4644
'Path W4645
SFTOF3D
SFTON3D P042
MOVJ C00746 BC00746 VJ=100.00  +MOVJ EC00746 VJ=100.00
SMOVL C00747 BC00747 V=800.0  +MOVJ EC00747
SMOVL C00748 BC00748 V=150.0 PL=0  +MOVJ EC00748
ARCON
SMOVL C00749 BC00749 V=11.7  +MOVJ EC00749
ARCOF
SMOVL C00750 BC00750 V=800.0  +MOVJ EC00750
SMOVL C00751 BC00751 V=1000.0  +MOVJ EC00751
SFTOF3D
'EndPath W4645
'Path W4646
SFTOF3D
SFTON3D P042
MOVJ C00752 BC00752 VJ=100.00  +MOVJ EC00752 VJ=100.00
SMOVL C00753 BC00753 V=800.0  +MOVJ EC00753
SMOVL C00754 BC00754 V=150.0 PL=0  +MOVJ EC00754
ARCON
SMOVL C00755 BC00755 V=11.7  +MOVJ EC00755
ARCOF
SMOVL C00756 BC00756 V=800.0  +MOVJ EC00756
SMOVL C00757 BC00757 V=1000.0  +MOVJ EC00757
SFTOF3D
'EndPath W4646
'3
MOVJ C00758 BC00758 VJ=100.00  +MOVJ EC00758 VJ=100.00
MOVJ C00759 BC00759 VJ=100.00  +MOVJ EC00759 VJ=100.00
'Path W4647
SFTOF3D
SFTON3D P044
MOVJ C00760 BC00760 VJ=100.00  +MOVJ EC00760 VJ=100.00
SMOVL C00761 BC00761 V=800.0  +MOVJ EC00761
SMOVL C00762 BC00762 V=150.0 PL=0  +MOVJ EC00762
ARCON
SMOVL C00763 BC00763 V=11.7  +MOVJ EC00763
ARCOF
SMOVL C00764 BC00764 V=800.0  +MOVJ EC00764
SMOVL C00765 BC00765 V=1000.0  +MOVJ EC00765
SFTOF3D
'EndPath W4647
'Path W4648
SFTOF3D
SFTON3D P046
MOVJ C00766 BC00766 VJ=100.00  +MOVJ EC00766 VJ=100.00
SMOVL C00767 BC00767 V=800.0  +MOVJ EC00767
SMOVL C00768 BC00768 V=150.0 PL=0  +MOVJ EC00768
MACRO1 MJ#(0) ARGF14
ARCON
SMOVL C00769 BC00769 V=11.7  +MOVJ EC00769
ARCOF
SMOVL C00770 BC00770 V=800.0  +MOVJ EC00770
SMOVL C00771 BC00771 V=1000.0  +MOVJ EC00771
SFTOF3D
'EndPath W4648
MOVJ C00772 BC00772 VJ=100.00  +MOVJ EC00772 VJ=100.00
MOVJ C00773 BC00773 VJ=100.00  +MOVJ EC00773 VJ=100.00
END
